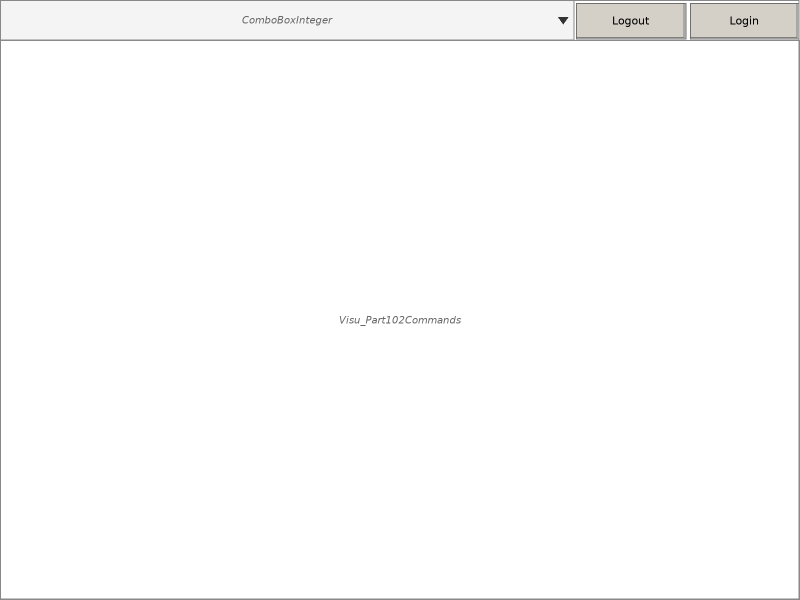
VISUALIZATION Visu_DALICommissioning  // 800x600
    ComboBoxInteger (0,0 574x40), variable: DALI_Commissioning.nSelectedDialog, input disabled if: DALI_Commissioning.bDisableComboBox, text list: 'TextList_Dialogs'
    Frame (0,40 800x560), frame switch variable: DALI_Commissioning.nSelectedDialog
        shows Visu_Part102Commands()
        shows Visu_Part102Parameters()
        shows Visu_Part102Addressing()
        shows Visu_Part102Groups()
        shows Visu_Part102Scenes()
        shows Visu_Part102MemoryBank()
        shows Visu_Part102SetFading()
        shows Visu_Part207Status()
        shows Visu_Part103Parameters()
        shows Visu_Part103Addressing()
        shows Visu_Part301PushButton()
        shows Visu_Part302AbsoluteInputDevice()
        shows Visu_Part303OccupancySensor()
        shows Visu_Part304LightSensor()
        shows Visu_Part300GenericDevice()
        shows Visu_Part103MemoryBank()
        shows Visu_KL6821Configuration()
    Button (690,3 109x36), "Login"
        OnMouseClick: VisuUserMgmt Type=Login
    Button (576,3 110x36), "Logout"
        OnMouseClick: VisuUserMgmt Type=Logout
END_VISUALIZATION

(* stored: Version 1.1.0.1, ProductVersion 3.1.4024.12
   Visu Visu_DALICommissioning: Id {a4bff0e3-4c5d-4f71-bb1e-168f27d09256} *)
